TYPE ST_UN_Machine_Hmi :
STRUCT
	// Local var
	fbHmiAlarmCollector		: FB_HMI_AlarmCollector;

END_STRUCT
END_TYPE

(* stored: Version 1.1.0.1, ProductVersion 3.1.4026.13
   DUT ST_UN_Machine_Hmi: Id {a5a17497-9654-44ef-bb9f-cbe16e8154ff} *)
